// TIA Portal V17 export
// export: Created 2026-04-13T11:12:04.8483814Z, ExportSetting WithDefaults, DisplayName Totally Integrated Automation Portal, DisplayVersion V17 Update 4, DisplayName TIA Portal Openness, DisplayVersion V17 Update 4, DisplayName TIA Portal Version Control Interface, DisplayVersion V17, DisplayName SINAMICS Startdrive Advanced, DisplayVersion V17, DisplayName SINAMICS Startdrive G130, G150, S120, S150, SINAMICS MV, S210, DisplayVersion V17, DisplayName SINAMICS Startdrive G110M, G120, G120C, G120D, G120P, G115D, DisplayVersion V17, DisplayName STEP 7 Professional, DisplayVersion V17 Update 4, DisplayName STEP 7 Safety, DisplayVersion V17, DisplayName WinCC Professional, DisplayVersion V17 Update 4
FUNCTION_BLOCK "A8-通信心跳"   // FB31, SCL
{ S7_Optimized_Access := 'TRUE' }
VERSION : 0.1
// stored: AutoNumber true, IsIECCheckEnabled false, IsRetainMemResEnabled false, MemoryReserve 100, SetENOAutomatically false, UDAEnableTagReadback false
   VAR_INPUT
      XH信号超时报警 : Real := 120.0;   // SB设备写读与创造写对比,如果不同超时,即判断报警
   END_VAR
   VAR_OUTPUT
      设备未通信报警 : Bool;
   END_VAR
   VAR_IN_OUT
      SB设备写读 : Real;
      SB设备写 : Real;
      SB设备写检测 : Real;
   END_VAR
   VAR RETAIN
      MC脉冲切换时间 : Real := 20.0;   // 给写信号+1,创造不同，10秒切换一次
   END_VAR
   VAR
      XH信号不同超时报警 : Real := 120.0;   // SB设备写读与创造写对比,如果不同超时,即判断报警
      XH信号相同超时报警 : Real := 120.0;   // SB设备写读与创造写对比,如果相同超时,即判断报警
      TON1 { S7_SetPoint := 'True'} : TON_TIME;
      TON1ET { S7_SetPoint := 'True'} : Time;
      TON2 : TON_TIME;
      TON2ET { S7_SetPoint := 'True'} : Time;
      LS设备通延辅助1 { S7_SetPoint := 'True'} : Bool;
      LS设备通延辅助2 : Bool;
      LS通信脉冲读1 : Bool;
      LS通信脉冲读2 : Bool;
      LS设备读温比较 : Real;
      T1S : TON_TIME;
      YC1 { S7_SetPoint := 'True'} : Real;
   END_VAR
   VAR_TEMP
      "m" : Int;
   END_VAR
BEGIN
   IF "FirstScan" THEN
       RESET_TIMER(#TON1);
       RESET_TIMER(#TON2);
       #LS设备通延辅助1 := 0;
       #LS设备通延辅助2 := 0;
   END_IF;

   #XH信号不同超时报警:=#XH信号超时报警;
   #XH信号相同超时报警 := #XH信号超时报警;
   #MC脉冲切换时间 := 20;

   IF #T1S.Q AND #YC1<#MC脉冲切换时间 THEN
       #YC1 := #YC1 + 1;
   END_IF;

   IF #YC1 >= #MC脉冲切换时间 THEN
       #YC1 := 0;
   END_IF;

   IF #YC1 <= (#MC脉冲切换时间 - 10) THEN

       #LS通信脉冲读1 := 1;
       #LS通信脉冲读2 := 0;
   ELSE
       #LS通信脉冲读1 := 0;
       #LS通信脉冲读2 := 1;
   END_IF;

   IF #LS通信脉冲读1 THEN
       //冷水
       #LS设备读温比较 := #SB设备写读;
       #SB设备写检测 := #SB设备写 + 0.1;
       #TON1(IN := (ABS(#LS设备读温比较) <> ABS(#SB设备写检测)),
             PT := DINT_TO_TIME(REAL_TO_DINT(#XH信号不同超时报警 * 1000.0)),
             Q => #LS设备通延辅助1,
             ET => #TON1ET);

      #TON2(IN := (ABS(#LS设备读温比较) = ABS(#SB设备写检测)),
             PT := DINT_TO_TIME(REAL_TO_DINT(#XH信号相同超时报警 * 1000.0)),
             Q => #LS设备通延辅助2,
             ET => #TON2ET);

   END_IF;

   IF #LS通信脉冲读2 AND NOT #LS通信脉冲读1 THEN
       #SB设备写检测 := #SB设备写;
   END_IF;

   IF #LS设备通延辅助1 OR #LS设备通延辅助2  THEN
       #设备未通信报警 := 1;
   ELSE
       #设备未通信报警 := 0;
   END_IF;

   #T1S(IN := NOT #T1S.Q,
       PT := T#1S);
END_FUNCTION_BLOCK
